// TwinCAT 3 PLC project Anker_WUCampus
// ProgramVersion: 3.1.4023.0
// libraries:
//   EfficientIO Communicator, * (EfficientIO)
//   Lynus Energy Basic, * (Lynus AG)
//   Lynus Persistent Data V1, * (Lynus AG)
//   Lynus Standards, * (Lynus AG)
//   Tc2_BABasic, * (Beckhoff Automation GmbH)
//   Tc2_Standard, * (Beckhoff Automation GmbH)
//   Tc2_System, * (Beckhoff Automation GmbH)
//   Tc2_Utilities, * (Beckhoff Automation GmbH)
//   Tc3_IotBase, * (Beckhoff Automation GmbH)
//   Tc3_JsonXml, * (Beckhoff Automation GmbH)
//   Tc3_Module, * (Beckhoff Automation GmbH)
// project tree:
//   / FastTask.TcTTO (not stored), MiddleTask.TcTTO, SlowTask.TcTTO (not stored)
//   FBs/ FB_Shelly_Pro1PM.TcPOU (not stored), FB_Shelly_Pro1PM_Helper.TcPOU (not stored), FB_TimeSwitch.TcPOU (not stored), FB_TimeSwitch_V2.TcPOU (not stored)
//   POUs/ prg5513EMS.TcPOU, prgComEffIO.TcPOU, prg5513Con.TcPOU, prg5513Grid.TcPOU, prgPersistent.TcPOU, prgRWEffIO.TcPOU, prgVarEffIO.TcPOU (not stored), prg_SystemTime.TcPOU (not stored)
// real-time tasks:
//   TASK FastTask: cycle T#5ms, priority 19, ADS port 350
//   TASK MiddleTask: cycle T#10ms, priority 20, ADS port 351
//   TASK SlowTask: cycle T#20ms, priority 21, ADS port 352
// I/O:
//   DEVICE Device 1 (Beckhoff CCAT)
//   DEVICE Device 2 (CX-BK)
//     Box 1 (CX-BK)
// variable links:
//   Anker_WUCampus/Anker_WUCampus Instance <-> Device 2 (CX-BK)/Box 1 (CX-BK)
//     MiddleTask Inputs/prg5513Grid.fbGrid1.fbKL3403.byStateCH1 <-> Term 3 (KL3403)/Channel 1/State
//     MiddleTask Inputs/prg5513Grid.fbGrid1.fbKL3403.byStateCH2 <-> Term 3 (KL3403)/Channel 2/State
//     MiddleTask Inputs/prg5513Grid.fbGrid1.fbKL3403.byStateCH3 <-> Term 3 (KL3403)/Channel 3/State
//     MiddleTask Inputs/prg5513Grid.fbGrid2.fbKL3403.byStateCH1 <-> Term 4 (KL3403)/Channel 1/State
//     MiddleTask Inputs/prg5513Grid.fbGrid2.fbKL3403.byStateCH2 <-> Term 4 (KL3403)/Channel 2/State
//     MiddleTask Inputs/prg5513Grid.fbGrid2.fbKL3403.byStateCH3 <-> Term 4 (KL3403)/Channel 3/State
//     MiddleTask Inputs/prg5513Grid.fbGrid1.fbKL3403.iDataInCH1 <-> Term 3 (KL3403)/Channel 1/Data In
//     MiddleTask Inputs/prg5513Grid.fbGrid1.fbKL3403.iDataInCH2 <-> Term 3 (KL3403)/Channel 2/Data In
//     MiddleTask Inputs/prg5513Grid.fbGrid1.fbKL3403.iDataInCH3 <-> Term 3 (KL3403)/Channel 3/Data In
//     MiddleTask Inputs/prg5513Grid.fbGrid2.fbKL3403.iDataInCH1 <-> Term 4 (KL3403)/Channel 1/Data In
//     MiddleTask Inputs/prg5513Grid.fbGrid2.fbKL3403.iDataInCH2 <-> Term 4 (KL3403)/Channel 2/Data In
//     MiddleTask Inputs/prg5513Grid.fbGrid2.fbKL3403.iDataInCH3 <-> Term 4 (KL3403)/Channel 3/Data In
//     MiddleTask Inputs/prg5513Grid.fbKBusState.uiKBusState_OUT <-> Inputs/State
//     MiddleTask Outputs/prg5513EMS.bQ1Switch <-> Term 2 (KL2408)/Channel 1/Output
//     MiddleTask Outputs/prg5513Grid.fbGrid1.fbKL3403.byCntrCH1 <-> Term 3 (KL3403)/Channel 1/Ctrl
//     MiddleTask Outputs/prg5513Grid.fbGrid1.fbKL3403.byCntrCH2 <-> Term 3 (KL3403)/Channel 2/Ctrl
//     MiddleTask Outputs/prg5513Grid.fbGrid1.fbKL3403.byCntrCH3 <-> Term 3 (KL3403)/Channel 3/Ctrl
//     MiddleTask Outputs/prg5513Grid.fbGrid2.fbKL3403.byCntrCH1 <-> Term 4 (KL3403)/Channel 1/Ctrl
//     MiddleTask Outputs/prg5513Grid.fbGrid2.fbKL3403.byCntrCH2 <-> Term 4 (KL3403)/Channel 2/Ctrl
//     MiddleTask Outputs/prg5513Grid.fbGrid2.fbKL3403.byCntrCH3 <-> Term 4 (KL3403)/Channel 3/Ctrl

CONFIGURATION Anker_WUCampus
    RESOURCE PLC ON TwinCAT3
        TASK MiddleTask(INTERVAL := T#10ms, PRIORITY := 20);
        PROGRAM prg5513Grid WITH MiddleTask : prg5513Grid;
        PROGRAM prgPersistent WITH MiddleTask : prgPersistent;
        PROGRAM prg5513Con WITH MiddleTask : prg5513Con;
        PROGRAM prg5513EMS WITH MiddleTask : prg5513EMS;
    END_RESOURCE
END_CONFIGURATION

// ---- POUs/prg5513Grid.TcPOU
PROGRAM prg5513Grid
VAR
	fbKBusState			: FB_K_Bus_State;
	lrPowerGrid			: LREAL;							//{#lynus.ag#()}
	lrCounterGrid		: LREAL;							//{#lynus.ag#()}
	// Grid1
	fbGrid1				: FB_EM_Beckhoff_KL3403;
	lrPowerGrid1		: LREAL;							//{#lynus.ag#()}
	lrCounterGrid1		: LREAL;							//{#lynus.ag#()}
	lrVoltageGrid1L1	: LREAL;							//{#lynus.ag#()}
	lrVoltageGrid1L2	: LREAL;							//{#lynus.ag#()}
	lrVoltageGrid1L3	: LREAL;							//{#lynus.ag#()}
	// Grid2
	fbGrid2				: FB_EM_Beckhoff_KL3403;
	lrPowerGrid2		: LREAL;							//{#lynus.ag#()}
	lrCounterGrid2		: LREAL;							//{#lynus.ag#()}
	lrVoltageGrid2L1	: LREAL;							//{#lynus.ag#()}
	lrVoltageGrid2L2	: LREAL;							//{#lynus.ag#()}
	lrVoltageGrid2L3	: LREAL;							//{#lynus.ag#()}
	uint_BusState	: UINT;									//{#lynus.ag#()}
END_VAR

//The mapping of this function must be linked with the K-Bus State in the E/A Part
fbKBusState(	uiKBusState_OUT=> , 
				b_Kbus_notOk=> , 
				word_ErrorCount=> );

//The mapping of this function must be linked with the KL3403 in the E/A Part
fbGrid1(
	bEnable:= TRUE, 
	bChannel1Invers:= FALSE,					//Invert power data when transformer are mounted upside down
	bChannel2Invers:= FALSE,
	bChannel3Invers:= FALSE,
	uiCurrentTransformerRatioL1:= 400, 		//Transformer ratio on the secondary side
	uiCurrentTransformerRatioL2:= 400, 
	uiCurrentTransformerRatioL3:= 400, 
	uiKBusState_IN:= fbKBusState.uiKBusState_OUT, 
	stDataEMPower=> , 
	stDataEMCounter=> , 
	stDataEMPowerRealTime=> , 
	stDataEMCounterRealTime=> , 
	diNrOfEM_OUT=> );

lrPowerGrid1 := fbGrid1.stDataEMPower.lrPowerTotal;
	lrCounterGrid1 := fbGrid1.stDataEMCounter.lrTotalCounterEnergy_Consumption;	
		lrVoltageGrid1L1 := fbGrid1.stDataEMPowerRealTime.lrVoltageL1N;
			lrVoltageGrid1L2 := fbGrid1.stDataEMPowerRealTime.lrVoltageL2N;
				lrVoltageGrid1L3 := fbGrid1.stDataEMPowerRealTime.lrVoltageL3N;


fbGrid2(
	bEnable:= TRUE, 
	bChannel1Invers:= FALSE,					//Invert power data when transformer are mounted upside down
	bChannel2Invers:= FALSE,
	bChannel3Invers:= FALSE,
	uiCurrentTransformerRatioL1:= 400, 		//Transformer ratio on the secondary side
	uiCurrentTransformerRatioL2:= 400, 
	uiCurrentTransformerRatioL3:= 400, 
	uiKBusState_IN:= fbKBusState.uiKBusState_OUT, 
	stDataEMPower=> , 
	stDataEMCounter=> , 
	stDataEMPowerRealTime=> , 
	stDataEMCounterRealTime=> , 
	diNrOfEM_OUT=> );

lrPowerGrid2 := fbGrid2.stDataEMPower.lrPowerTotal;
	lrCounterGrid2 := fbGrid2.stDataEMCounter.lrTotalCounterEnergy_Consumption;	
		lrVoltageGrid2L1 := fbGrid2.stDataEMPowerRealTime.lrVoltageL1N;
			lrVoltageGrid2L2 := fbGrid2.stDataEMPowerRealTime.lrVoltageL2N;
				lrVoltageGrid2L3 := fbGrid2.stDataEMPowerRealTime.lrVoltageL3N;
lrPowerGrid := 	lrPowerGrid1 + lrPowerGrid2;
			
uint_BusState := fbKbusState.uiKBusState_OUT;

END_PROGRAM

// ---- POUs/prgPersistent.TcPOU
PROGRAM prgPersistent
VAR
	fbUSV		: FB_WritePersistentData_CX81xx;
END_VAR

fbUSV(
	eSaveModeData:= eUSVSaveMode.eSaveWhenPowerfail, 
	bLoadPersistentDataOk=> , 
	bPowerFailDetect=> , 
	bError=> , 
	bySaveProcess=> , 
	dwStorageLast24h=> , 
	udiErrorCode=> );

prg_SystemTime();

END_PROGRAM

// ---- POUs/prg5513Con.TcPOU
PROGRAM prg5513Con
VAR
	// Shelly1: 
//	fbShelly1				:	FB_Shelly_Pro1PM;
	lrS1P1Power				:	LREAL;			//{#lynus.ag#()}
	lrS1P1Power_kW			:	LREAL;			//{#lynus.ag#()}
	lrS1P1Voltage			:	LREAL;			//{#lynus.ag#()}
	lrS1P1Energy			:	LREAL;			//{#lynus.ag#()}
	lrS1P1Temperature		:	LREAL;			//{#lynus.ag#()}
	bS1P1On					:	BOOL;			//{#lynus.ag#()}
	bS1P1Off				:	BOOL;			//{#lynus.ag#()}
	bS1P1Switch				:	BOOL;			//{#lynus.ag#()}
	
	// Shelly2: 
//	fbShelly2				:	FB_Shelly_Pro1PM;
	lrS2P1Power				:	LREAL;			//{#lynus.ag#()}
	lrS2P1Power_kW			:	LREAL;			//{#lynus.ag#()}
	lrS2P1Voltage			:	LREAL;			//{#lynus.ag#()}
	lrS2P1Energy			:	LREAL;			//{#lynus.ag#()}
	lrS2P1Temperature		:	LREAL;			//{#lynus.ag#()}
	bS2P1On					:	BOOL;			//{#lynus.ag#()}
	bS2P1Off				:	BOOL;			//{#lynus.ag#()}
	bS2P1Switch				:	BOOL;			//{#lynus.ag#()}
	
	// Shelly3: 
//	fbShelly3				:	FB_Shelly_Pro1PM;
	lrS3P1Power				:	LREAL;			//{#lynus.ag#()}
	lrS3P1Power_kW			:	LREAL;			//{#lynus.ag#()}
	lrS3P1Voltage			:	LREAL;			//{#lynus.ag#()}
	lrS3P1Energy			:	LREAL;			//{#lynus.ag#()}
	lrS3P1Temperature		:	LREAL;			//{#lynus.ag#()}
	bS3P1On					:	BOOL;			//{#lynus.ag#()}
	bS3P1Off				:	BOOL;			//{#lynus.ag#()}
	bS3P1Switch				:	BOOL;			//{#lynus.ag#()}
	
	// Shelly4: 
//	fbShelly4				:	FB_Shelly_Pro1PM;
	lrS4P1Power				:	LREAL;			//{#lynus.ag#()}
	lrS4P1Power_kW			:	LREAL;			//{#lynus.ag#()}
	lrS4P1Voltage			:	LREAL;			//{#lynus.ag#()}
	lrS4P1Energy			:	LREAL;			//{#lynus.ag#()}
	lrS4P1Temperature		:	LREAL;			//{#lynus.ag#()}
	bS4P1On					:	BOOL;			//{#lynus.ag#()}
	bS4P1Off				:	BOOL;			//{#lynus.ag#()}
	bS4P1Switch				:	BOOL;			//{#lynus.ag#()}
	
	// Shelly5: 
//	fbShelly5				:	FB_Shelly_Pro1PM;
	lrS5P1Power				:	LREAL;			//{#lynus.ag#()}
	lrS5P1Power_kW			:	LREAL;			//{#lynus.ag#()}
	lrS5P1Voltage			:	LREAL;			//{#lynus.ag#()}
	lrS5P1Energy			:	LREAL;			//{#lynus.ag#()}
	lrS5P1Temperature		:	LREAL;			//{#lynus.ag#()}
	bS5P1On					:	BOOL;			//{#lynus.ag#()}
	bS5P1Off				:	BOOL;			//{#lynus.ag#()}
	bS5P1Switch				:	BOOL;			//{#lynus.ag#()}
	
	// Other
	lrRemainPower_kW		:	LREAL;			//{#lynus.ag#()}
	
	// state maschine for GET requests
	str_Array_IPs			: array[1..30] of STRING(15);			//arrays for IPs
	int_State: INT;
	
	int_Multiplier_1 			:INT:=1;								// multilpier received values, =2 when external fuse is on, was at the beginning
	int_Multiplier_2 			:INT:=2;								// multilpier received values, =2 when external fuse is on, was at the beginning
	int_Multiplier_3 			:INT:=2;								// multilpier received values, =2 when external fuse is on, was at the beginning
	int_Multiplier_4 			:INT:=1;								// multilpier received values, =2 when external fuse is on, was at the beginning
	int_Multiplier_5 			:INT:=1;								// multilpier received values, =2 when external fuse is on, was at the beginning

	int_TimeoutCounter: ARRAY[1..30] OF INT;	
	int_SuccessCounter: ARRAY[1..30] OF INT;	
	int_ErrorCounter: ARRAY[1..30] OF INT;
	ton_wait: Ton;
	fbShelly				:	ARRAY[1..20] OF FB_Shelly_Pro1PM;
	f_Trig_Busy				:	ARRAY[1..20] OF f_trig;
	m_Error_HTTP: BOOL;							//{#lynus.ag#()}
END_VAR

CASE int_State OF
	0: 		// Init State
	
	// define IPs
	str_Array_IPs[1]	:='10.55.13.131';
	str_Array_IPs[2]	:='10.55.13.132';
	str_Array_IPs[3]	:='10.55.13.133';
	str_Array_IPs[4]	:='10.55.13.134';		
	str_Array_IPs[5]	:='10.55.13.135';
	str_Array_IPs[6]	:='';
	str_Array_IPs[7]	:='';
	str_Array_IPs[8]	:='';
	str_Array_IPs[9]	:='';
	str_Array_IPs[10]	:='';
	str_Array_IPs[11]	:='';
	str_Array_IPs[12]	:='';
	str_Array_IPs[13]	:='';
	str_Array_IPs[14]	:='';
	fbShelly[1].sHostname:= str_Array_IPs[1];
	fbShelly[2].sHostname:= str_Array_IPs[2];
	fbShelly[3].sHostname:= str_Array_IPs[3];
	fbShelly[4].sHostname:= str_Array_IPs[4];
	fbShelly[5].sHostname:= str_Array_IPs[5];
 
	
	// =2 for the beginning when bypass fuse is on
	int_Multiplier_1:=1;
	int_Multiplier_2:=2;
	int_Multiplier_3:=2;
	int_Multiplier_4:=1;
	int_Multiplier_5:=1;

	IF str_Array_IPs[1] <> '' THEN
		int_State :=1;
	END_IF
		
	1: 		// request
	
		fbShelly[int_State].bStart:= TRUE;
		fbShelly[int_State].bOnP1:= bS1P1On;
		fbShelly[int_State].bOffP1:= bS1P1Off;
	
		f_Trig_Busy[int_State](CLK :=fbShelly[int_State].bBusy);
			
		// go to next state
		IF f_Trig_Busy[int_State].Q  AND NOT fbShelly[int_State].bError THEN	
			int_SuccessCounter[int_State]	:= int_SuccessCounter[int_State]+1;
			lrS1P1Power 	:= 	fbShelly[int_State].lrpowerP1 * int_Multiplier_1;
			lrS1P1Energy 	:= 	fbShelly[int_State].lrenergyP1 * int_Multiplier_1;
			lrS1P1Voltage	:=	fbShelly[int_State].lrvoltageP1; 
			lrS1P1Temperature :=fbShelly[int_State].lrTemperatureP1;
			bS1P1Switch		:=	fbShelly[int_State].bStateP1;
		ELSIF  f_Trig_Busy[int_State].Q  AND fbShelly[int_State].bError THEN
			int_ErrorCounter[int_State]	:= int_ErrorCounter[int_State]+1;
		END_IF
		IF 	int_state < 20 AND str_Array_IPs[int_State+1] <> '' AND f_Trig_Busy[int_State].Q  THEN	
			fbShelly[int_State].bStart		:= FALSE;
			int_State := int_State+1;
		ELSIF  (str_Array_IPs[int_State+1] = '' OR int_state > 20) AND f_Trig_Busy[int_State].Q THEN
			fbShelly[int_State].bStart		:= FALSE;
			int_State := 100;			// wait state for new run
		END_IF		
	
	2: 		// request
	
		fbShelly[int_State].bStart:= TRUE;
		fbShelly[int_State].bOnP1:= bS2P1On;
		fbShelly[int_State].bOffP1:= bS2P1Off;
	
		f_Trig_Busy[int_State](CLK :=fbShelly[int_State].bBusy);
			
		// go to next state
		IF f_Trig_Busy[int_State].Q  AND NOT fbShelly[int_State].bError THEN	
			int_SuccessCounter[int_State]	:= int_SuccessCounter[int_State]+1;
			lrS2P1Power 	:= 	fbShelly[int_State].lrpowerP1 * int_Multiplier_2;
			lrS2P1Energy 	:= 	fbShelly[int_State].lrenergyP1 * int_Multiplier_2;
			lrS2P1Temperature :=fbShelly[int_State].lrTemperatureP1;
			lrS2P1Voltage	:=	fbShelly[int_State].lrvoltageP1; 
			bS2P1Switch		:=	fbShelly[int_State].bStateP1;
		ELSIF  f_Trig_Busy[int_State].Q  AND fbShelly[int_State].bError THEN
			int_ErrorCounter[int_State]	:= int_ErrorCounter[int_State]+1;
		END_IF
		IF 	int_state < 20 AND str_Array_IPs[int_State+1] <> '' AND f_Trig_Busy[int_State].Q  THEN	
			fbShelly[int_State].bStart		:= FALSE;
			int_State := int_State+1;
		ELSIF  (str_Array_IPs[int_State+1] = '' OR int_state > 20) AND f_Trig_Busy[int_State].Q THEN
			fbShelly[int_State].bStart		:= FALSE;
			int_State := 100;			// wait state for new run
		END_IF	
		
	3: 		// request
		fbShelly[int_State].bStart:= TRUE;
		fbShelly[int_State].bOnP1:= bS3P1On;
		fbShelly[int_State].bOffP1:= bS3P1Off;
	
		f_Trig_Busy[int_State](CLK :=fbShelly[int_State].bBusy);
			
		// go to next state
		IF f_Trig_Busy[int_State].Q  AND NOT fbShelly[int_State].bError THEN	
			int_SuccessCounter[int_State]	:= int_SuccessCounter[int_State]+1;
			lrS3P1Power 	:= 	fbShelly[int_State].lrpowerP1 * int_Multiplier_3;
			lrS3P1Energy 	:= 	fbShelly[int_State].lrenergyP1 * int_Multiplier_3;
			lrS3P1Temperature :=fbShelly[int_State].lrTemperatureP1;
			lrS3P1Voltage	:=	fbShelly[int_State].lrvoltageP1; 
			bS3P1Switch		:=	fbShelly[int_State].bStateP1;
		ELSIF  f_Trig_Busy[int_State].Q  AND fbShelly[int_State].bError THEN
			int_ErrorCounter[int_State]	:= int_ErrorCounter[int_State]+1;
		END_IF
		IF 	int_state < 20 AND str_Array_IPs[int_State+1] <> '' AND f_Trig_Busy[int_State].Q  THEN	
			fbShelly[int_State].bStart		:= FALSE;
			int_State := int_State+1;
		ELSIF  (str_Array_IPs[int_State+1] = '' OR int_state > 20) AND f_Trig_Busy[int_State].Q THEN
			fbShelly[int_State].bStart		:= FALSE;
			int_State := 100;			// wait state for new run
		END_IF	
	4: 		// request
	
		fbShelly[int_State].bStart:= TRUE;
		fbShelly[int_State].bOnP1:= bS4P1On;
		fbShelly[int_State].bOffP1:= bS4P1Off;
	
		f_Trig_Busy[int_State](CLK :=fbShelly[int_State].bBusy);
		// go to next state
		IF f_Trig_Busy[int_State].Q  AND NOT fbShelly[int_State].bError THEN	
			int_SuccessCounter[int_State]	:= int_SuccessCounter[int_State]+1;
			lrS4P1Power 	:= 	fbShelly[int_State].lrpowerP1 * int_Multiplier_4;
			lrS4P1Energy 	:= 	fbShelly[int_State].lrenergyP1 * int_Multiplier_4;
			lrS4P1Temperature :=fbShelly[int_State].lrTemperatureP1;
			lrS4P1Voltage	:=	fbShelly[int_State].lrvoltageP1; 
			bS4P1Switch		:=	fbShelly[int_State].bStateP1;
		ELSIF  f_Trig_Busy[int_State].Q  AND fbShelly[int_State].bError THEN
			int_ErrorCounter[int_State]	:= int_ErrorCounter[int_State]+1;
		END_IF
		IF 	int_state < 20 AND str_Array_IPs[int_State+1] <> '' AND f_Trig_Busy[int_State].Q  THEN	
			fbShelly[int_State].bStart		:= FALSE;
			int_State := int_State+1;
		ELSIF  (str_Array_IPs[int_State+1] = '' OR int_state > 20) AND f_Trig_Busy[int_State].Q THEN
			fbShelly[int_State].bStart		:= FALSE;
			int_State := 100;			// wait state for new run
		END_IF
		
	5: 		// request
	
		fbShelly[int_State].bStart:= TRUE;
		fbShelly[int_State].bOnP1:= bS5P1On;
		fbShelly[int_State].bOffP1:= bS5P1Off;
	
		f_Trig_Busy[int_State](CLK :=fbShelly[int_State].bBusy);
			
		// go to next state
		IF f_Trig_Busy[int_State].Q  AND NOT fbShelly[int_State].bError THEN	
			int_SuccessCounter[int_State]	:= int_SuccessCounter[int_State]+1;
			lrS5P1Power 	:= 	fbShelly[int_State].lrpowerP1 * int_Multiplier_5;
			lrS5P1Energy 	:= 	fbShelly[int_State].lrenergyP1 * int_Multiplier_5;
			lrS5P1Temperature :=fbShelly[int_State].lrTemperatureP1;
			lrS5P1Voltage	:=	fbShelly[int_State].lrvoltageP1; 
			bS5P1Switch		:=	fbShelly[int_State].bStateP1;
		ELSIF  f_Trig_Busy[int_State].Q  AND fbShelly[int_State].bError THEN
			int_ErrorCounter[int_State]	:= int_ErrorCounter[int_State]+1;
		END_IF
		IF 	int_state < 20 AND str_Array_IPs[int_State+1] <> '' AND f_Trig_Busy[int_State].Q  THEN	
			fbShelly[int_State].bStart		:= FALSE;
			int_State := int_State+1;
		ELSIF  (str_Array_IPs[int_State+1] = '' OR int_state > 20) AND f_Trig_Busy[int_State].Q THEN
			fbShelly[int_State].bStart		:= FALSE;
			int_State := 100;			// wait state for new run
		END_IF	
	
	100:		// wait state
	ton_wait.IN :=TRUE;
	IF ton_wait.Q THEN
		ton_wait.IN :=FALSE;
//		IF NOT fbShelly[1].bError THEN
			int_State := 1;
//		ELSIF fbShelly[1].bError AND prg_SystemTime.structSystemTime.wHour=4 AND prg_SystemTime.structSystemTime.wMinute>45 THEN
//			int_State := 1;
//		ELSE
//			int_State := 3;
//		END_IF
	END_IF		
END_CASE


// Shelly communication

fbShelly[1](tDelayRequest:= T#0S, );
fbShelly[2](tDelayRequest:= T#0S, );
fbShelly[3](tDelayRequest:= T#0S, );
fbShelly[4](tDelayRequest:= T#0S, );
fbShelly[5](tDelayRequest:= T#0S, );


// wait
ton_wait(PT:=T#3S);


// re-calc to kW
lrS1P1Power_kW := lrS1P1Power / 1000;
lrS2P1Power_kW := lrS2P1Power / 1000;
lrS3P1Power_kW := lrS3P1Power / 1000;
lrS4P1Power_kW := lrS4P1Power / 1000;
lrS5P1Power_kW := lrS5P1Power / 1000;
				
// Other
lrRemainPower_kW := LIMIT(0, prg5513Grid.lrPowerGrid - (lrS1P1Power_kW + lrS2P1Power_kW + lrS3P1Power_kW + lrS4P1Power_kW + lrS5P1Power_kW), 999999);
	
// on / off commands from EMS
// Kühlpult Shelly 1
fbShelly[1].bEnableControl := TRUE;		// prg5513EMS.FB_TimeSwitch_CoolingCounter.b_Enable;
IF prg5513EMS.FB_TimeSwitch_CoolingCounter.b_Output_On AND NOT fbShelly[1].bStateP1 THEN
	bS1P1On :=TRUE;
ELSE
	bS1P1On := FALSE;
END_IF
IF NOT prg5513EMS.FB_TimeSwitch_CoolingCounter.b_Output_On AND fbShelly[1].bStateP1 THEN
	bS1P1Off :=TRUE;
ELSE
	bS1P1Off := FALSE;
END_IF
// Boiler Shelly 4
fbShelly[4].bEnableControl := TRUE;		// prg5513EMS.FB_TimeSwitch_Boiler.b_Enable;
IF prg5513EMS.FB_TimeSwitch_Boiler.b_Output_On AND NOT fbShelly[4].bStateP1 THEN
	bS4P1On :=TRUE;
ELSE
	bS4P1On := FALSE;
END_IF
IF NOT prg5513EMS.FB_TimeSwitch_Boiler.b_Output_On AND fbShelly[4].bStateP1 THEN
	bS4P1Off :=TRUE;
ELSE
	bS4P1Off := FALSE;
END_IF

// Klima Shelly 5
fbShelly[5].bEnableControl := true;		// prg5513EMS.FB_TimeSwitch_AC.b_Enable;
IF prg5513EMS.FB_TimeSwitch_AC.b_Output_On AND NOT fbShelly[5].bStateP1 THEN
	bS5P1On :=TRUE;
ELSE
	bS5P1On := FALSE;
END_IF
IF NOT prg5513EMS.FB_TimeSwitch_AC.b_Output_On AND fbShelly[5].bStateP1 THEN
	bS5P1Off :=TRUE;
ELSE
	bS5P1Off := FALSE;
END_IF

// error bit to cloud 

m_Error_HTTP := fbShelly[1].bError OR fbShelly[4].bError OR fbShelly[5].bError;

END_PROGRAM

// ---- POUs/prg5513EMS.TcPOU
PROGRAM prg5513EMS
VAR
	//coffee machine relay
	bQ1Switch	AT%Q*	: BOOL;						//{#lynus.ag#()}
	
	FB_TimeSwitch_Coffee: FB_TimeSwitch_V2;	
	FB_TimeSwitch_AC: FB_TimeSwitch_V2;				// Shelly 5
	FB_TimeSwitch_CoolingCounter: FB_TimeSwitch_V2;	// Shelly 1
	FB_TimeSwitch_Boiler: FB_TimeSwitch_V2;			// Shelly 4
	FB_TimeSwitch_Outside: FB_TimeSwitch_V2;		// no outside light at WU campus
	

	b_Coffee_Manual_On: BOOL;						//{#lynus.ag#()}
	b_Coffee_Manual_Off: BOOL;						//{#lynus.ag#()}
	b_AC_Manual_On: BOOL;							//{#lynus.ag#()}
	b_AC_Manual_Off: BOOL;							//{#lynus.ag#()}
	b_CoolingCounter_Manual_On: BOOL;				//{#lynus.ag#()}
	b_CoolingCounter_Manual_Off: BOOL;				//{#lynus.ag#()}
	b_Boiler_Manual_On: BOOL;						//{#lynus.ag#()}
	b_Boiler_Manual_Off: BOOL;						//{#lynus.ag#()}
	b_Outside_Manual_On: BOOL;						//{#lynus.ag#()}
	b_Outside_Manual_Off: BOOL;						//{#lynus.ag#()}

	fbCalcSunriseSunset   		: FB_CalcSunriseSunset;
	todSunrise            		: TOD;
	todSunset             		: TOD;
	fb_GetTimeZoneInfo	:FB_GetTimeZoneInformation;
	b_firstCycle: BOOL;
	RS_Outsidelight: RS;
	r_trig_on: R_trig;
	r_trig_off: R_trig;

	b_Status_CoffeeMaschine: BOOL;					//{#lynus.ag#()}
END_VAR
VAR PERSISTENT
// opening hours	
	byte_MoFr_Open_Hour		:BYTE;								//{#lynus.ag#()}
	byte_MoFr_Open_Minute	:BYTE;								//{#lynus.ag#()}
	byte_MoFr_Close_Hour	:BYTE;								//{#lynus.ag#()}
	byte_MoFr_Close_Minute	:BYTE;								//{#lynus.ag#()}
	byte_Sa_Open_Hour		:BYTE;								//{#lynus.ag#()}
	byte_Sa_Open_Minute		:BYTE;								//{#lynus.ag#()}
	byte_Sa_Close_Hour		:BYTE;								//{#lynus.ag#()}
	byte_Sa_Close_Minute	:BYTE;								//{#lynus.ag#()}
	byte_So_Open_Hour		:BYTE;								//{#lynus.ag#()}
	byte_So_Open_Minute		:BYTE;								//{#lynus.ag#()}
	byte_So_Close_Hour		:BYTE;								//{#lynus.ag#()}
	byte_So_Close_Minute	:BYTE;								//{#lynus.ag#()}
	
// offset coffeemaschine in hours			
	b_Enable_Control_Coffee		:BOOL;								//{#lynus.ag#()}
	real_Coffee_Offset_Start	:REAL;								//{#lynus.ag#()}
	real_Coffee_Offset_Stop		:REAL;								//{#lynus.ag#()}

// offset AC in hours			
	b_Enable_Control_AC			:BOOL;								//{#lynus.ag#()}
	real_AC_Offset_Start		:REAL;								//{#lynus.ag#()}
	real_AC_Offset_Stop			:REAL;								//{#lynus.ag#()}
	
// offset CoolingCounter in hours			
	b_Enable_Control_CoolingCounter		:BOOL;								//{#lynus.ag#()}
	real_CoolingCounter_Offset_Start		:REAL;								//{#lynus.ag#()}
	real_CoolingCounter_Offset_Stop		:REAL;								//{#lynus.ag#()}

// offset Boiler Cooler in hours			
	b_Enable_Control_Boiler	:BOOL;								//{#lynus.ag#()}
	real_Boiler_Offset_Start	:REAL;								//{#lynus.ag#()}
	real_Boiler_Offset_Stop	:REAL;								//{#lynus.ag#()}


END_VAR

FB_TimeSwitch_Coffee(
	b_Enable:= b_Enable_Control_Coffee, 
	b_StatusOn:= NOT bQ1Switch, 
	structSystemTime:=prg_SystemTime.structSystemTime , 
	byte_MoFr_Open_Hour:= byte_MoFr_Open_Hour , 
	byte_MoFr_Open_Minute:= byte_MoFr_Open_Minute, 
	byte_MoFr_Close_Hour:= byte_MoFr_Close_Hour , 
	byte_MoFr_Close_Minute:= byte_MoFr_Close_Minute, 
	byte_Sa_Open_Hour:= byte_Sa_Open_Hour, 
	byte_Sa_Open_Minute:= byte_Sa_Open_Minute , 
	byte_Sa_Close_Hour:= byte_Sa_Close_Hour , 
	byte_Sa_Close_Minute:= byte_Sa_Close_Minute, 
	byte_So_Open_Hour:= byte_So_Open_Hour, 
	byte_So_Open_Minute:= byte_So_Open_Minute, 
	byte_So_Close_Hour:= byte_So_Close_Hour, 
	byte_So_Close_Minute:= byte_So_Close_Minute, 
	real_Offset_Start:= real_Coffee_Offset_Start , 
	real_Offset_Stop:= real_Coffee_Offset_Stop , 
	b_On_Manual:= b_Coffee_Manual_On, 
	b_Off_Manual:= b_Coffee_Manual_Off, 
	b_Output_On=> , 
	b_Error=> );
IF NOT FB_TimeSwitch_Coffee.b_Output_On THEN
	bQ1Switch := TRUE;
ELSIF FB_TimeSwitch_Coffee.b_Output_On THEN
	bQ1Switch := FALSE;
END_IF
b_Status_CoffeeMaschine := NOT bQ1Switch;

FB_TimeSwitch_AC(
	b_Enable:= b_Enable_Control_AC, 
	b_StatusOn:= prg5513CON.fbShelly[5].bStateP1, 
	structSystemTime:= prg_SystemTime.structSystemTime , 
	byte_MoFr_Open_Hour:= byte_MoFr_Open_Hour , 
	byte_MoFr_Open_Minute:= byte_MoFr_Open_Minute, 
	byte_MoFr_Close_Hour:= byte_MoFr_Close_Hour , 
	byte_MoFr_Close_Minute:= byte_MoFr_Close_Minute, 
	byte_Sa_Open_Hour:= byte_Sa_Open_Hour, 
	byte_Sa_Open_Minute:= byte_Sa_Open_Minute , 
	byte_Sa_Close_Hour:= byte_Sa_Close_Hour , 
	byte_Sa_Close_Minute:= byte_Sa_Close_Minute, 
	byte_So_Open_Hour:= byte_So_Open_Hour, 
	byte_So_Open_Minute:= byte_So_Open_Minute, 
	byte_So_Close_Hour:= byte_So_Close_Hour, 
	byte_So_Close_Minute:= byte_So_Close_Minute, 
	real_Offset_Start:= real_AC_Offset_Start , 
	real_Offset_Stop:= real_AC_Offset_Stop , 
	b_On_Manual:= b_AC_Manual_On, 
	b_Off_Manual:= b_AC_Manual_Off, 
	b_Output_On=> , 
	b_Error=> );

FB_TimeSwitch_CoolingCounter(
	b_Enable:= b_Enable_Control_CoolingCounter, 
	b_StatusOn:= prg5513CON.fbShelly[1].bStateP1, 
	structSystemTime:= prg_SystemTime.structSystemTime , 
	byte_MoFr_Open_Hour:= byte_MoFr_Open_Hour , 
	byte_MoFr_Open_Minute:= byte_MoFr_Open_Minute, 
	byte_MoFr_Close_Hour:= byte_MoFr_Close_Hour , 
	byte_MoFr_Close_Minute:= byte_MoFr_Close_Minute, 
	byte_Sa_Open_Hour:= byte_Sa_Open_Hour, 
	byte_Sa_Open_Minute:= byte_Sa_Open_Minute , 
	byte_Sa_Close_Hour:= byte_Sa_Close_Hour , 
	byte_Sa_Close_Minute:= byte_Sa_Close_Minute, 
	byte_So_Open_Hour:= byte_So_Open_Hour, 
	byte_So_Open_Minute:= byte_So_Open_Minute, 
	byte_So_Close_Hour:= byte_So_Close_Hour, 
	byte_So_Close_Minute:= byte_So_Close_Minute, 
	real_Offset_Start:= real_CoolingCounter_Offset_Start , 
	real_Offset_Stop:= real_CoolingCounter_Offset_Stop , 
	b_On_Manual:= b_CoolingCounter_Manual_On, 
	b_Off_Manual:= b_CoolingCounter_Manual_Off, 
	b_Output_On=> , 
	b_Error=> );

FB_TimeSwitch_Boiler(
	b_Enable:= b_Enable_Control_Boiler, 
	b_StatusOn:= prg5513CON.fbShelly[4].bStateP1, 
	structSystemTime:= prg_SystemTime.structSystemTime , 
	byte_MoFr_Open_Hour:= byte_MoFr_Open_Hour , 
	byte_MoFr_Open_Minute:= byte_MoFr_Open_Minute, 
	byte_MoFr_Close_Hour:= byte_MoFr_Close_Hour , 
	byte_MoFr_Close_Minute:= byte_MoFr_Close_Minute, 
	byte_Sa_Open_Hour:= byte_Sa_Open_Hour, 
	byte_Sa_Open_Minute:= byte_Sa_Open_Minute , 
	byte_Sa_Close_Hour:= byte_Sa_Close_Hour , 
	byte_Sa_Close_Minute:= byte_Sa_Close_Minute, 
	byte_So_Open_Hour:= byte_So_Open_Hour, 
	byte_So_Open_Minute:= byte_So_Open_Minute, 
	byte_So_Close_Hour:= byte_So_Close_Hour, 
	byte_So_Close_Minute:= byte_So_Close_Minute, 
	real_Offset_Start:= real_Boiler_Offset_Start , 
	real_Offset_Stop:= real_Boiler_Offset_Stop , 
	b_On_Manual:= b_Boiler_Manual_On, 
	b_Off_Manual:= b_Boiler_Manual_Off, 
	b_Output_On=> , 
	b_Error=> );

// not needed for WU Campus, no outside light. 
// calculate sunset / sunrise
// find out the time details
fb_GetTimeZoneInfo(
	sNetID:= '', 
	bExecute:= prg_SystemTime.structSystemTime.wHour = 4 OR NOT b_firstCycle, 
	tTimeout:= T#5S, 
	bBusy=> , 
	bError=> , 
	nErrID=> , 
	tzID=> , 
	tzInfo=> );
b_firstCycle := TRUE;

fbCalcSunriseSunset(
	fDegreeOfLongitude := 16.3731,   (* Longitude of Vienna *)
	fDegreeOfLatitude := 48.2083,   (* Latitude of Vienna*)
	fReferenceMeridian := SEL( fb_GetTimeZoneInfo.tzID = eTimeZoneID_Daylight ,15,30),  (* Central European Time 15 Winter Timer / 30 Summer Time *)
	dCurrentDate := DT_TO_DATE(SYSTEMTIME_TO_Dt (prg_SystemTime.structSystemTime)),
	todSunrise => todSunrise,
	todSunset => todSunset);

r_trig_on (clk := FB_TimeSwitch_Outside.b_Output_On AND DT_TO_TOD(systemtime_to_dt(prg_SystemTime.structSystemTime))< (todSunrise +  T#1H) );
r_trig_off (clk := NOT FB_TimeSwitch_Outside.b_Output_On);

RS_Outsidelight(	Set := r_trig_on.Q OR ((todSunset - T#2H) =  DT_TO_TOD(systemtime_to_dt(prg_SystemTime.structSystemTime)) AND FB_TimeSwitch_Outside.b_Output_On) ,
					Reset1 := r_trig_off.Q OR ((todSunrise +  T#1H)= DT_TO_TOD(systemtime_to_dt(prg_SystemTime.structSystemTime))),
					Q1 => );

END_PROGRAM

// ---- POUs/prgComEffIO.TcPOU
PROGRAM prgComEffIO
VAR
	fbCom		: FB_MqttCommunicator;
END_VAR

fbCom(
	bConnect:= TRUE, 
	sUserName:= '485eb9d2-182c-41ae-9a36-0282f763bd0c', 
	sUserPassword:= '8ad9d088-a47d-4765-a173-1fddc80662af', 
	eSavePositionCertificate:= eSavePositionOnPLC.ePostionHardDisk, 
	bConnected=> , 
	bError=> , 
	hrErrorCode=> , 
	eConnectionState=> , 
	eErrorMessage_Out=> );

END_PROGRAM

// ---- POUs/prgRWEffIO.TcPOU
PROGRAM prgRWEffIO
VAR
	fbRW1		: FB_ReadWrite_V2;
END_VAR

fbRW1(
	eUploadType:= 3, // Change + 5 min Intervall  
	bBusy=> , 
	bError=> , 
	udiErrorCodeOut=> , 
	eErrorReadWrite_Out=> );

END_PROGRAM
